// Mitsubishi GX Works2 project: 0730-1   PLC: Q02/Q02H

PROGRAM MAIN
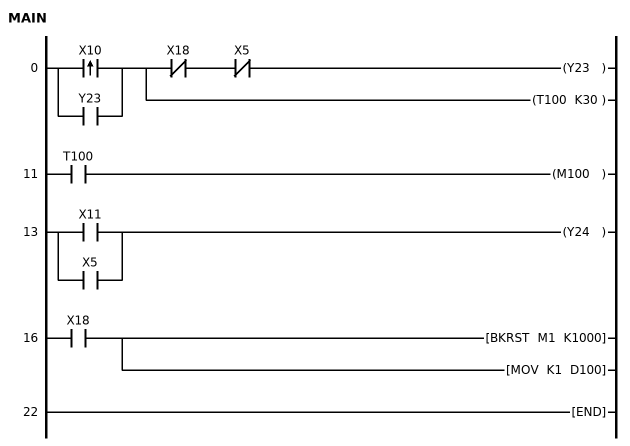
0     LDP     X10
      OR      Y23
      MPS
      ANI     X18
      ANI     X5
      OUT     Y23
      MPP
      OUT     T100 K30
11    LD      T100
      OUT     M100
13    LD      X11
      OR      X5
      OUT     Y24
16    LD      X18
      BKRST   M1 K1000
      MOV     K1 D100
22    END
END_PROGRAM

PROGRAM HMI
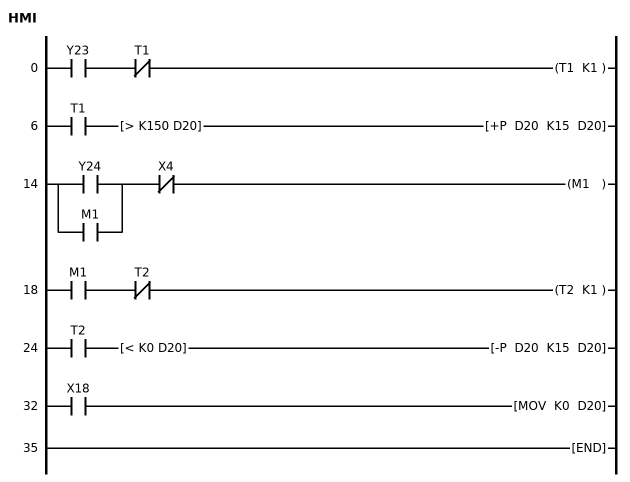
0     LD      Y23
      ANI     T1
      OUT     T1 K1
6     LD      T1
      AND>    K150 D20
      +P      D20 K15 D20
14    LD      Y24
      OR      M1
      ANI     X4
      OUT     M1
18    LD      M1
      ANI     T2
      OUT     T2 K1
24    LD      T2
      AND<    K0 D20
      -P      D20 K15 D20
32    LD      X18
      MOV     K0 D20
35    END
END_PROGRAM

PROGRAM ERROR
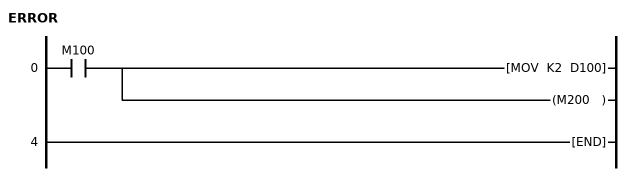
0     LD      M100
      MOV     K2 D100
      OUT     M200
4     END
END_PROGRAM
